PROGRAM Lift_Raise_and_Lower
VAR
	LiftRaiseRequest: BOOL; // Logic bit to request transfer move forward towards lift bed.
	LiftLowerRequest: BOOL; // Logic bit to request transfer move reverse towards home switch
	ReadyToRaise:BOOL; // Logic bit to indicate ready to lift
	ReadyToLower:BOOL; // Logic bit to indicate ready to lower
	OpenTransferClampRequest:BOOL; // Logic bit to request transfer clamp open
	CloseTransferClampRequest:BOOL; // Logic bit to request transfer clamp close
	TransferFwdRequest: BOOL; // Logic bit to request transfer move forward towards lift bed.
	TransferRevRequest: BOOL; // Logic bit to request transfer move reverse towards home switch
	RibsReadyForPickup:BOOL; // Hoist is up and ribs have been cut to lenght, waiting for gripper to acknowledge pick up
	
END_VAR

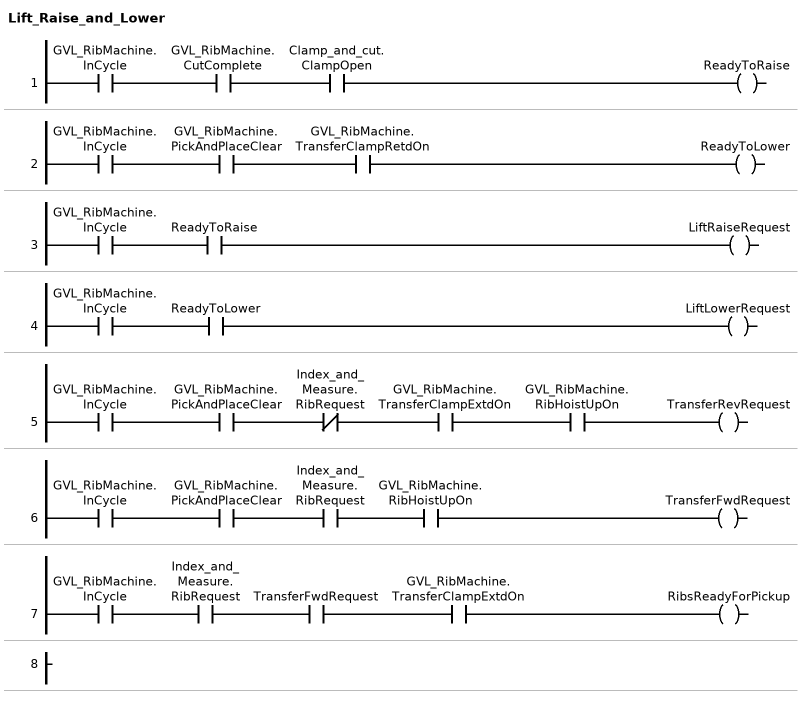
// NETWORK 1
ReadyToRaise := GVL_RibMachine.InCycle AND GVL_RibMachine.CutComplete AND Clamp_and_cut.ClampOpen;

// NETWORK 2
ReadyToLower := GVL_RibMachine.InCycle AND GVL_RibMachine.PickAndPlaceClear AND GVL_RibMachine.TransferClampRetdOn;

// NETWORK 3
LiftRaiseRequest := GVL_RibMachine.InCycle AND ReadyToRaise;

// NETWORK 4
LiftLowerRequest := GVL_RibMachine.InCycle AND ReadyToLower;

// NETWORK 5
TransferRevRequest := GVL_RibMachine.InCycle AND GVL_RibMachine.PickAndPlaceClear AND NOT Index_and_Measure.RibRequest AND GVL_RibMachine.TransferClampExtdOn AND GVL_RibMachine.RibHoistUpOn;

// NETWORK 6
TransferFwdRequest := GVL_RibMachine.InCycle AND GVL_RibMachine.PickAndPlaceClear AND Index_and_Measure.RibRequest AND GVL_RibMachine.RibHoistUpOn;

// NETWORK 7
RibsReadyForPickup := GVL_RibMachine.InCycle AND Index_and_Measure.RibRequest AND TransferFwdRequest AND GVL_RibMachine.TransferClampExtdOn;

// NETWORK 8

END_PROGRAM

(* stored: Version 1.1.0.1, ProductVersion 3.1.4024.12
   POU Lift_Raise_and_Lower: Id {b7a7f776-65c0-4696-85b6-8d5cc845276e}, SpecialFunc None *)
